{attribute 'GeneratedUsingTerminal: EK1960-0000-0021'}
{attribute addProperty BoxType "EK1960-0000-0021"}
{attribute addProperty Id "FSOEAT %Q*FSOE_3E4279E151"}
{attribute addProperty CRC "3624411961"}
{attribute addProperty Size "51"}
TYPE FSoE_Outputs_D8082339 :
STRUCT
	{attribute addProperty Name "FSOE"}
	FSOE AT %Q* : FSOE_3E4279E1;
END_STRUCT
END_TYPE

(* stored: Version 1.2.0.0, ProductVersion 3.1.4024.9
   DUT FSoE_Outputs_D8082339: Id {6e1ca369-668e-4c24-b251-59dd96bc7f96} *)
